// TIA Portal V17 export
// export: Created 2021-09-22T11:25:08.8348708Z, ExportSetting WithDefaults, DisplayName Totally Integrated Automation Portal, DisplayVersion V17, DisplayName TIA Portal Openness, DisplayVersion V17, DisplayName TIA Portal Version Control Interface, DisplayVersion V17, DisplayName SINAMICS Startdrive Advanced, DisplayVersion V17, DisplayName SINAMICS Startdrive G130, G150, S120, S150, SINAMICS MV, S210, DisplayVersion V17, DisplayName SINAMICS Startdrive G110M, G120, G120C, G120D, G120P, G115D, DisplayVersion V17, DisplayName STEP 7 Professional, DisplayVersion V17, DisplayName STEP 7 Safety, DisplayVersion V17, DisplayName WinCC Advanced / Unified PC, DisplayVersion V17
TYPE "Motor_type"
// stored: IsFailsafeCompliant false
   STRUCT
      Cmd : "MotorCmd_type";
      Status : "MotorStatus_type";
      Setting : "MotorSetting_type";
      Control { S7_SetPoint := 'True'} : "MotorControl_type";
   END_STRUCT;
END_TYPE
